FUNCTION F_Concat5_Large : LongString
VAR_IN_OUT CONSTANT
   sOne : LongString;
   sTwo : LongString;
   sThree : LongString;
   sFour : LongString;
   sFive : LongString;
END_VAR
VAR
   str : LongString;
END_VAR

str := F_Concat4_Large(sTwo, sThree, sFour, sFive);
F_Concat5_Large :=
   F_ConcatLarge(
      sOne,
      str
   );

END_FUNCTION

(* stored: Version 1.1.0.1, ProductVersion 3.1.4024.9
   POU F_Concat5_Large: Id {ca0d4fe3-5327-4cb8-beb5-b6aa0c1c934b}, SpecialFunc None *)
